// TIA Portal V15 export
// export: Created 2018-12-10T18:36:41.6560857Z, ExportSetting WithDefaults, WithReadOnly, DisplayName Totally Integrated Automation Portal, DisplayVersion V15 Update 2, DisplayName TIA Portal Openness, DisplayVersion V15 Update 2, DisplayName STEP 7 Professional, DisplayVersion V15 Update 2, DisplayName STEP 7 Safety, DisplayVersion V15, DisplayName WinCC Professional, DisplayVersion V15 Update 2, DisplayName SIMATIC Visualization Architect, DisplayVersion V15 Update 1
DATA_BLOCK "DB_ACTIONS_SEQUENCENAME"   // DB171
TITLE = Action sequence / Aktionen Ablaufkette
{ S7_Optimized_Access := 'FALSE' }
VERSION : 0.1
// stored: AutoNumber true, CodeModifiedDate 2016-11-16T08:22:55.1691627Z, CompileDate 2018-02-20T10:24:41.1893532Z, CreationDate 2016-12-16T08:19:32.7526446Z, DBAccessibleFromOPCUA true, InterfaceModifiedDate 2016-09-07T23:28:40.167814Z, IsConsistent true, IsKnowHowProtected false, IsOnlyStoredInLoadMemory false, IsPLCDB false, IsWriteProtectedInAS false, ModifiedDate 2018-01-29T16:41:39.5932916Z, ParameterModified 2016-09-07T23:28:40.167814Z, StructureModified 2016-09-07T23:28:40.167814Z
   VAR RETAIN
      A_INI { ExternalAccessible := 'False'; ExternalVisible := 'False'; ExternalWritable := 'False'} : Bool;   // Initialstep / Anfangsposition Station leer
      A_GRD { ExternalAccessible := 'False'; ExternalVisible := 'False'; ExternalWritable := 'False'} : Bool;   // check home position / Prüfe Homeposition
      A_FM { ExternalAccessible := 'False'; ExternalVisible := 'False'; ExternalWritable := 'False'} : Bool;   // End / Ende
      A_Dummy { ExternalAccessible := 'False'; ExternalVisible := 'False'; ExternalWritable := 'False'} : Bool;   // Dummy step / Leerschritt
      A_stop_before_process { ExternalAccessible := 'False'; ExternalVisible := 'False'; ExternalWritable := 'False'} : Bool;   // Stop before process welding/HSN / Halt vor Prozeß Schweißen / HSN
      A_stop_after_process { ExternalAccessible := 'False'; ExternalVisible := 'False'; ExternalWritable := 'False'} : Bool;   // Stop after process welding/HSN / Halt nach Prozeß Schweißen / HSN
   END_VAR
BEGIN
END_DATA_BLOCK
